Omron Sysmac Studio project test_mqtt (Sysmac Studio 1.45.1.64010, StandardProject)

# Controller new_Controller_0: NX1P2-9024DT version 1.40
Task PrimaryTask (priority 4, period or condition 2000): Program0
Library MQTT 0.44.98f 0.44.98 (contents left out)

PROGRAM Program0
VAR
    Connect_broker : BOOL;
    CLIENT(MQTT) : MQTT\MQTTClient;
    HostBroker : STRING[256];
    ServerPortBroker : UINT;
    ClientIDBroker : STRING[64];
    BufferBroker : MQTT\ClientBuffer;
END_VAR

(* Section Section0: ladder, written here as Structured Text *)

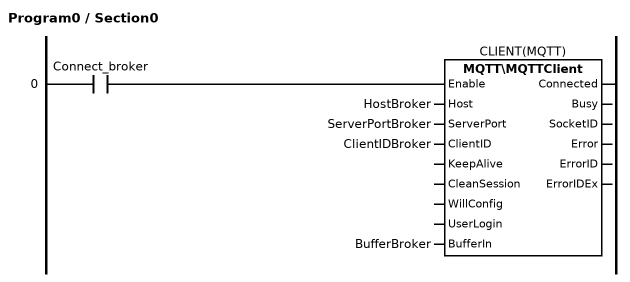
(* Rung 0 *)
CLIENT(MQTT)(Enable := Connect_broker, Host := HostBroker, ServerPort := ServerPortBroker, ClientID := ClientIDBroker, BufferIn := BufferBroker);
END_PROGRAM